// TwinCAT 3 PLC project txi_hxr_motion
// Title: txi-hxr-motion
// Company: SLAC
// ProjectVersion: 2.0.0
// ProgramVersion: 3.1.4024.12
// libraries:
//   LCLS General, * (SLAC)
//   lcls-twincat-motion, * (SLAC)
//   lcls-twincat-physics, * (SLAC)
//   lcls2-cc-lib, * (SLAC)
//   PMPS, * (SLAC - LCLS)
//   Tc2_MC2, * (Beckhoff Automation GmbH)
//   Tc2_Standard, * (Beckhoff Automation GmbH)
//   Tc2_System, * (Beckhoff Automation GmbH)
//   Tc3_Module, * (Beckhoff Automation GmbH)
// project tree:
//   GVLs/ GVL.TcGVL, Main.TcGVL
//   Version/ Global_Version.TcGVL
//   / PlcTask.TcTTO
//   POUs/ PRG_AL1L1_L2SI.TcPOU, PRG_IM2L1_PPM.TcPOU, PRG_01_PLCTASK.TcPOU, PRG_PMPS.TcPOU, PRG_SL3L1_SCATTER.TcPOU, PRG_TXI_PM.TcPOU
//   POUs/temp/ FB_SLITS.TcPOU (not stored), FB_SLITS_POWER.TcPOU (not stored), FB_SLITS_SCATTER.TcPOU (not stored)
// real-time tasks:
//   TASK PlcTask: cycle T#10ms, priority 20, ADS port 350
// motion (NC):
//   TASK NC-Task 1 SAF: cycle T#2ms, priority 4, ADS port 501
//   TASK NC-Task 1 SVB: cycle T#10ms, priority 8, ADS port 511
//   AXIS IM2L1-PPM-MMS (id 2)
//     Dynamic: AccelerationMaximum=200, DecelerationMaximum=200, Acceleration=200, Deceleration=200, Jerk=1000, DelayTime=0.004
//     Velo: Maximum=65
//     MotionControl: Enable=true, Range=0.0005, Time=1
//     TargetPosControl: Range=0.01, Time=1
//     OtherSettings: AllowMotionCmdToSlave=true
//     encoder EncType=29
//       EncPara: ScaleFactorNumerator=5e-05, Offset=-214686.941, MaxCount=#xffffffff, ReferenceSystem=1
//         SoftEndMinControl: Enable=true, Range=-95
//         SoftEndMaxControl: Enable=true, Range=-5
//         Inc: RefSoftSyncMask=#x0000ffff
//     drive DrvType=24
//       Analog: VeloReferenz=100, ScaleFactorActTorque=0.1
//       TimeComp: TaskDelayCycles=1
//     controller CtrType=2
//       CtrPara: PriorControlFactor=1
//         PosDiffControl: Range=10, Time=0.1
//         PID: PosKp=10, PosExtKp=0.01, PosExtVelo=0.0005, DeadBandPosition=0.0001
//         Observer: BandWidth=20
//   AXIS SL3L1-BOTTOM-MMS (id 3)
//   AXIS SL3L1-NORTH-MMS (id 5) // C:\Github\lcls-plc-tmo-motion\plc-tmo-motion\_Config\NC\Axes\SL2K4-NORTH-M25.xti
//     Velo: RefSearch=0.2, RefSync=0.05, Maximum=2.2
//     OtherSettings: AllowMotionCmdToSlave=true
//     encoder EncType=4
//       EncPara: Inverse=true, MaxCount=#x0000ffff
//         SoftEndMinControl: Enable=true, Range=-30.81
//         SoftEndMaxControl: Enable=true
//         Inc: RefSoftSyncMask=#x0000ffff
//     drive DrvType=24
//       Analog: VeloReferenz=2, ScaleFactorActTorque=0.1
//       TimeComp: TaskDelayCycles=1
//     controller CtrType=1
//       CtrPara: PriorControlFactor=1
//         Observer: BandWidth=20
//   AXIS SL3L1-SOUTH-MMS (id 6) // C:\Github\lcls-plc-tmo-motion\plc-tmo-motion\_Config\NC\Axes\SL2K4-SOUTH-M26.xti
//     Velo: RefSearch=0.2, RefSync=0.05, Maximum=2.2
//     OtherSettings: AllowMotionCmdToSlave=true
//     encoder EncType=4
//       EncPara: MaxCount=#x0000ffff
//         SoftEndMinControl: Enable=true, Range=-30.52
//         SoftEndMaxControl: Enable=true
//         Inc: RefSoftSyncMask=#x0000ffff
//     drive DrvType=24
//       Analog: VeloReferenz=2, ScaleFactorActTorque=0.1
//       TimeComp: TaskDelayCycles=1
//     controller CtrType=1
//       CtrPara: PriorControlFactor=1
//         Observer: BandWidth=20
//   AXIS SL3L1-TOP-MMS (id 4) // C:\Github\lcls-plc-tmo-motion\plc-tmo-motion\_Config\NC\Axes\SL2K4-TOP-M24.xti
//     Velo: RefSearch=0.2, RefSync=0.05, Maximum=2.2
//     PositionAreaControl: Range=0.5
//     TargetPosControl: Range=0.1
//     OtherSettings: AllowMotionCmdToSlave=true
//     encoder EncType=4
//       EncPara: Inverse=true, MaxCount=#x0000ffff
//         SoftEndMinControl: Enable=true, Range=-30.91
//         SoftEndMaxControl: Enable=true
//         Inc: RefSoftSyncMask=#x0000ffff
//     drive DrvType=24
//       Analog: VeloReferenz=2, ScaleFactorActTorque=0.1
//       TimeComp: TaskDelayCycles=1
//     controller CtrType=1
//       CtrPara: PriorControlFactor=1
//         PosDiffControl: Range=0.5
//         Observer: BandWidth=20
//   AXIS AL1L1-L2SI-MMS (id 1)
//     Dynamic: AccelerationMaximum=200, DecelerationMaximum=200, Acceleration=200, Deceleration=200, Jerk=500, DelayTime=0.004
//     Velo: Maximum=10
//     TargetPosControl: Range=0.002, Time=2
//     OtherSettings: AllowMotionCmdToSlave=true
//     encoder EncType=29
//       EncPara: ScaleFactorNumerator=5e-05, Offset=-214686.941, MaxCount=#xffffffff, ReferenceSystem=1
//         SoftEndMinControl: Enable=true, Range=-94
//         SoftEndMaxControl: Enable=true, Range=-37
//         Inc: RefSoftSyncMask=#x0000ffff
//     drive DrvType=24
//       Analog: VeloReferenz=100, ScaleFactorActTorque=0.1
//       TimeComp: TaskDelayCycles=1
//     controller CtrType=2
//       CtrPara: PriorControlFactor=1
//         PosDiffControl: Range=1
//         PID: PosKp=20, PosExtKp=1, PosExtVelo=0.1, DeadBandPosition=0.002
//         Observer: BandWidth=20
// I/O:
//   DEVICE Device 1 (EtherCAT), AmsNetId 172.21.136.31.2.1
//     R17-DRL-03 (EK1200) [EK1200-5000 EtherCAT Power supply (2A E-Bus)]
//       Term 8 (EL6070) [EL6070 1Ch. Licensing-Terminal]
//       Term 9 (EL2202) [EL2202 2Ch. Dig. Output 24V, 0.5A]
//       Term 10 (EL6695) [EL6695 EtherCAT Bridge terminal (Primary)]
//       Term 11 (EK1122) [EK1122 2 port EtherCAT junction]
//       Term 12 (EK1110)
//     100H1-L1S01-DRL-02 (EK1100) [EK1100 EtherCAT Coupler (2A E-Bus)]
//       E1 (EK1122) [EK1122 2 port EtherCAT junction]
//         AL1L1-L2SI (EK1100) [EK1100 EtherCAT Coupler (2A E-Bus)]
//           AL1L1-EL7041 [EL7041 1Ch. Stepper motor output stage (50V, 5A)]
//           AL1L1-EL5042 [EL5042 2Ch. BiSS-C Encoder]
//           AL1L1-EL2004 [EL2004 4Ch. Dig. Output 24V, 0.5A]
//           AL1L1-EL4004 [EL4004 4Ch. Ana. Output 0-10V, 12bit]
//           AL1L1-EL9011
//         IM2L1-PPM (EK1100) [EK1100 EtherCAT Coupler (2A E-Bus)]
//           IM2L1-EL7041 [EL7041 1Ch. Stepper motor output stage (50V, 5A)]
//           IM2L1-EL5042 [EL5042 2Ch. BiSS-C Encoder]
//           IM2L1-EL2004
//           IM2L1-EL3314 [EL3314 4Ch. Ana. Input Thermocouple (TC)]
//           IM2L1-EL3052 [EL3052 2Ch. Ana. Input 4-20mA]
//           IM2L1-EL3062 [EL3062 2Ch. Ana. Input 0-10V]
//           IM2L1-EL4004
//           IM2L1-EL9011
//       E2 (EK1122) [EK1122 2 port EtherCAT junction]
//         SL3L1-SCATTER (EK1100) [EK1100 EtherCAT Coupler (2A E-Bus)]
//           SL3L1-EL7031-E1 [EL7031 1Ch. Stepper motor output stage (24V, 1.5A)]
//           SL3L1-EL5101-E2 [EL5101 1Ch. Inc. Encoder 5V]
//           SL3L1-EL7031-E3 [EL7031 1Ch. Stepper motor output stage (24V, 1.5A)]
//           SL3L1-EL5101-E4 [EL5101 1Ch. Inc. Encoder 5V]
//           SL3L1-EL7031-E5 [EL7031 1Ch. Stepper motor output stage (24V, 1.5A)]
//           SL3L1-EL5101-E6
//           SL3L1-EL7031-E7 [EL7031 1Ch. Stepper motor output stage (24V, 1.5A)]
//           SL3L1-EL5101-E8
//           SL3L1-EL9011-E9
//       Term 33 (EK1110) [EK1110 EtherCAT extension]
//     TXI Power Meter (EK1100) [EK1100 EtherCAT Coupler (2A E-Bus)]
//       PM-EL3064
//       Term 70 (EK1122) [EK1122 2 port EtherCAT junction]
//       Term 74 (EL9011) [EL9011 End Terminal]
// variable links:
//   (this object) <-> Device 1 (EtherCAT)/100H1-L1S01-DRL-02 (EK1100)/E1 (EK1122)/IM2L1-PPM (EK1100)/IM2L1-EL5042
//     Enc/Inputs/In/nComState @bit 1 <-> WcState/InputToggle
//     Enc/Inputs/In/nComState <-> WcState/WcState
//     Enc/Inputs/In/nDataIn1 <-> FB Inputs Channel 1/Position
//     Enc/Inputs/In/nState1 @bit 12 <-> FB Inputs Channel 1/Status/Diag
//     Enc/Inputs/In/nState1 @bit 1 <-> FB Inputs Channel 1/Status/Error
//     Enc/Inputs/In/nState1 @bit 14 <-> FB Inputs Channel 1/Status/Input cycle counter
//     Enc/Inputs/In/nState1 @bit 2 <-> FB Inputs Channel 1/Status/Ready
//     Enc/Inputs/In/nState1 @bit 13 <-> FB Inputs Channel 1/Status/TxPDO State
//     Enc/Inputs/In/nState1 <-> FB Inputs Channel 1/Status/Warning
//   (this object) <-> Device 1 (EtherCAT)/100H1-L1S01-DRL-02 (EK1100)/E1 (EK1122)/IM2L1-PPM (EK1100)/IM2L1-EL7041
//     Drive/Inputs/In/nState1 @bit 3 <-> STM Status/Status/Error
//     Drive/Inputs/In/nState1 @bit 5 <-> STM Status/Status/Moving negative
//     Drive/Inputs/In/nState1 @bit 4 <-> STM Status/Status/Moving positive
//     Drive/Inputs/In/nState1 @bit 1 <-> STM Status/Status/Ready
//     Drive/Inputs/In/nState1 <-> STM Status/Status/Ready to enable
//     Drive/Inputs/In/nState1 @bit 6 <-> STM Status/Status/Torque reduced
//     Drive/Inputs/In/nState1 @bit 2 <-> STM Status/Status/Warning
//     Drive/Inputs/In/nState2 @bit 3 <-> STM Status/Status/Digital input 1
//     Drive/Inputs/In/nState2 @bit 4 <-> STM Status/Status/Digital input 2
//     Drive/Inputs/In/nState2 @bit 5 <-> STM Status/Status/Sync error
//     Drive/Inputs/In/nState2 @bit 7 <-> STM Status/Status/TxPDO Toggle
//     Drive/Inputs/In/nState4 @bit 1 <-> WcState/InputToggle
//     Drive/Inputs/In/nState4 <-> WcState/WcState
//     Drive/Outputs/Out/nCtrl1 <-> STM Control/Control/Enable
//     Drive/Outputs/Out/nCtrl1 @bit 2 <-> STM Control/Control/Reduce torque
//     Drive/Outputs/Out/nCtrl1 @bit 1 <-> STM Control/Control/Reset
//     Drive/Outputs/Out/nDataOut2[0] <-> STM Velocity/Velocity
//   (this object) <-> Device 1 (EtherCAT)/100H1-L1S01-DRL-02 (EK1100)/E2 (EK1122)/SL3L1-SCATTER (EK1100)/SL3L1-EL5101-E6
//     Enc/Inputs/In/nDataIn1[0] <-> ENC Status compact/Counter value
//     Enc/Inputs/In/nDataIn2[0] <-> ENC Status compact/Latch value
//     Enc/Inputs/In/nState1 @bit 4 <-> ENC Status compact/Status/Counter overflow
//     Enc/Inputs/In/nState1 @bit 3 <-> ENC Status compact/Status/Counter underflow
//     Enc/Inputs/In/nState1 @bit 7 <-> ENC Status compact/Status/Extrapolation stall
//     Enc/Inputs/In/nState1 <-> ENC Status compact/Status/Latch C valid
//     Enc/Inputs/In/nState1 @bit 1 <-> ENC Status compact/Status/Latch extern valid
//     Enc/Inputs/In/nState1 @bit 6 <-> ENC Status compact/Status/Open circuit
//     Enc/Inputs/In/nState1 @bit 2 <-> ENC Status compact/Status/Set counter done
//     Enc/Inputs/In/nState1 @bit 5 <-> ENC Status compact/Status/Status of input status
//     Enc/Inputs/In/nState2 @bit 4 <-> ENC Status compact/Status/Status of extern latch
//     Enc/Inputs/In/nState2 <-> ENC Status compact/Status/Status of input A
//     Enc/Inputs/In/nState2 @bit 1 <-> ENC Status compact/Status/Status of input B
//     Enc/Inputs/In/nState2 @bit 2 <-> ENC Status compact/Status/Status of input C
//     Enc/Inputs/In/nState2 @bit 3 <-> ENC Status compact/Status/Status of input gate
//     Enc/Inputs/In/nState2 @bit 5 <-> ENC Status compact/Status/Sync error
//     Enc/Inputs/In/nState2 @bit 6 <-> ENC Status compact/Status/TxPDO State
//     Enc/Inputs/In/nState2 @bit 7 <-> ENC Status compact/Status/TxPDO Toggle
//     Enc/Inputs/In/nState4 @bit 1 <-> WcState/InputToggle
//     Enc/Inputs/In/nState4 <-> WcState/WcState
//     Enc/Outputs/Out/nCtrl1 <-> ENC Control compact/Control/Enable latch C
//     Enc/Outputs/Out/nCtrl1 @bit 3 <-> ENC Control compact/Control/Enable latch extern on negative edge
//     Enc/Outputs/Out/nCtrl1 @bit 1 <-> ENC Control compact/Control/Enable latch extern on positive edge
//     Enc/Outputs/Out/nCtrl1 @bit 2 <-> ENC Control compact/Control/Set counter
//     Enc/Outputs/Out/nDataOut1[0] <-> ENC Control compact/Set counter value
//   (this object) <-> Device 1 (EtherCAT)/100H1-L1S01-DRL-02 (EK1100)/E2 (EK1122)/SL3L1-SCATTER (EK1100)/SL3L1-EL7031-E5
//     Drive/Inputs/In/nState1 @bit 3 <-> STM Status/Status/Error
//     Drive/Inputs/In/nState1 @bit 5 <-> STM Status/Status/Moving negative
//     Drive/Inputs/In/nState1 @bit 4 <-> STM Status/Status/Moving positive
//     Drive/Inputs/In/nState1 @bit 1 <-> STM Status/Status/Ready
//     Drive/Inputs/In/nState1 <-> STM Status/Status/Ready to enable
//     Drive/Inputs/In/nState1 @bit 6 <-> STM Status/Status/Torque reduced
//     Drive/Inputs/In/nState1 @bit 2 <-> STM Status/Status/Warning
//     Drive/Inputs/In/nState2 @bit 3 <-> STM Status/Status/Digital input 1
//     Drive/Inputs/In/nState2 @bit 4 <-> STM Status/Status/Digital input 2
//     Drive/Inputs/In/nState2 @bit 5 <-> STM Status/Status/Sync error
//     Drive/Inputs/In/nState2 @bit 7 <-> STM Status/Status/TxPDO Toggle
//     Drive/Inputs/In/nState4 @bit 1 <-> WcState/InputToggle
//     Drive/Inputs/In/nState4 <-> WcState/WcState
//     Drive/Outputs/Out/nCtrl1 <-> STM Control/Control/Enable
//     Drive/Outputs/Out/nCtrl1 @bit 2 <-> STM Control/Control/Reduce torque
//     Drive/Outputs/Out/nCtrl1 @bit 1 <-> STM Control/Control/Reset
//     Drive/Outputs/Out/nDataOut2[0] <-> STM Velocity/Velocity
//   (this object) <-> Device 1 (EtherCAT)/100H1-L1S01-DRL-02 (EK1100)/E2 (EK1122)/SL3L1-SCATTER (EK1100)/SL3L1-EL5101-E8
//     Enc/Inputs/In/nDataIn1[0] <-> ENC Status compact/Counter value
//     Enc/Inputs/In/nDataIn2[0] <-> ENC Status compact/Latch value
//     Enc/Inputs/In/nState1 @bit 4 <-> ENC Status compact/Status/Counter overflow
//     Enc/Inputs/In/nState1 @bit 3 <-> ENC Status compact/Status/Counter underflow
//     Enc/Inputs/In/nState1 @bit 7 <-> ENC Status compact/Status/Extrapolation stall
//     Enc/Inputs/In/nState1 <-> ENC Status compact/Status/Latch C valid
//     Enc/Inputs/In/nState1 @bit 1 <-> ENC Status compact/Status/Latch extern valid
//     Enc/Inputs/In/nState1 @bit 6 <-> ENC Status compact/Status/Open circuit
//     Enc/Inputs/In/nState1 @bit 2 <-> ENC Status compact/Status/Set counter done
//     Enc/Inputs/In/nState1 @bit 5 <-> ENC Status compact/Status/Status of input status
//     Enc/Inputs/In/nState2 @bit 4 <-> ENC Status compact/Status/Status of extern latch
//     Enc/Inputs/In/nState2 <-> ENC Status compact/Status/Status of input A
//     Enc/Inputs/In/nState2 @bit 1 <-> ENC Status compact/Status/Status of input B
//     Enc/Inputs/In/nState2 @bit 2 <-> ENC Status compact/Status/Status of input C
//     Enc/Inputs/In/nState2 @bit 3 <-> ENC Status compact/Status/Status of input gate
//     Enc/Inputs/In/nState2 @bit 5 <-> ENC Status compact/Status/Sync error
//     Enc/Inputs/In/nState2 @bit 6 <-> ENC Status compact/Status/TxPDO State
//     Enc/Inputs/In/nState2 @bit 7 <-> ENC Status compact/Status/TxPDO Toggle
//     Enc/Inputs/In/nState4 @bit 1 <-> WcState/InputToggle
//     Enc/Inputs/In/nState4 <-> WcState/WcState
//     Enc/Outputs/Out/nCtrl1 <-> ENC Control compact/Control/Enable latch C
//     Enc/Outputs/Out/nCtrl1 @bit 3 <-> ENC Control compact/Control/Enable latch extern on negative edge
//     Enc/Outputs/Out/nCtrl1 @bit 1 <-> ENC Control compact/Control/Enable latch extern on positive edge
//     Enc/Outputs/Out/nCtrl1 @bit 2 <-> ENC Control compact/Control/Set counter
//     Enc/Outputs/Out/nDataOut1[0] <-> ENC Control compact/Set counter value
//   (this object) <-> Device 1 (EtherCAT)/100H1-L1S01-DRL-02 (EK1100)/E2 (EK1122)/SL3L1-SCATTER (EK1100)/SL3L1-EL7031-E7
//     Drive/Inputs/In/nState1 @bit 3 <-> STM Status/Status/Error
//     Drive/Inputs/In/nState1 @bit 5 <-> STM Status/Status/Moving negative
//     Drive/Inputs/In/nState1 @bit 4 <-> STM Status/Status/Moving positive
//     Drive/Inputs/In/nState1 @bit 1 <-> STM Status/Status/Ready
//     Drive/Inputs/In/nState1 <-> STM Status/Status/Ready to enable
//     Drive/Inputs/In/nState1 @bit 6 <-> STM Status/Status/Torque reduced
//     Drive/Inputs/In/nState1 @bit 2 <-> STM Status/Status/Warning
//     Drive/Inputs/In/nState2 @bit 3 <-> STM Status/Status/Digital input 1
//     Drive/Inputs/In/nState2 @bit 4 <-> STM Status/Status/Digital input 2
//     Drive/Inputs/In/nState2 @bit 5 <-> STM Status/Status/Sync error
//     Drive/Inputs/In/nState2 @bit 7 <-> STM Status/Status/TxPDO Toggle
//     Drive/Inputs/In/nState4 @bit 1 <-> WcState/InputToggle
//     Drive/Inputs/In/nState4 <-> WcState/WcState
//     Drive/Outputs/Out/nCtrl1 <-> STM Control/Control/Enable
//     Drive/Outputs/Out/nCtrl1 @bit 2 <-> STM Control/Control/Reduce torque
//     Drive/Outputs/Out/nCtrl1 @bit 1 <-> STM Control/Control/Reset
//     Drive/Outputs/Out/nDataOut2[0] <-> STM Velocity/Velocity
//   (this object) <-> Device 1 (EtherCAT)/100H1-L1S01-DRL-02 (EK1100)/E2 (EK1122)/SL3L1-SCATTER (EK1100)/SL3L1-EL5101-E4
//     Enc/Inputs/In/nDataIn1[0] <-> ENC Status compact/Counter value
//     Enc/Inputs/In/nDataIn2[0] <-> ENC Status compact/Latch value
//     Enc/Inputs/In/nState1 @bit 4 <-> ENC Status compact/Status/Counter overflow
//     Enc/Inputs/In/nState1 @bit 3 <-> ENC Status compact/Status/Counter underflow
//     Enc/Inputs/In/nState1 @bit 7 <-> ENC Status compact/Status/Extrapolation stall
//     Enc/Inputs/In/nState1 <-> ENC Status compact/Status/Latch C valid
//     Enc/Inputs/In/nState1 @bit 1 <-> ENC Status compact/Status/Latch extern valid
//     Enc/Inputs/In/nState1 @bit 6 <-> ENC Status compact/Status/Open circuit
//     Enc/Inputs/In/nState1 @bit 2 <-> ENC Status compact/Status/Set counter done
//     Enc/Inputs/In/nState1 @bit 5 <-> ENC Status compact/Status/Status of input status
//     Enc/Inputs/In/nState2 @bit 4 <-> ENC Status compact/Status/Status of extern latch
//     Enc/Inputs/In/nState2 <-> ENC Status compact/Status/Status of input A
//     Enc/Inputs/In/nState2 @bit 1 <-> ENC Status compact/Status/Status of input B
//     Enc/Inputs/In/nState2 @bit 2 <-> ENC Status compact/Status/Status of input C
//     Enc/Inputs/In/nState2 @bit 3 <-> ENC Status compact/Status/Status of input gate
//     Enc/Inputs/In/nState2 @bit 5 <-> ENC Status compact/Status/Sync error
//     Enc/Inputs/In/nState2 @bit 6 <-> ENC Status compact/Status/TxPDO State
//     Enc/Inputs/In/nState2 @bit 7 <-> ENC Status compact/Status/TxPDO Toggle
//     Enc/Inputs/In/nState4 @bit 1 <-> WcState/InputToggle
//     Enc/Inputs/In/nState4 <-> WcState/WcState
//     Enc/Outputs/Out/nCtrl1 <-> ENC Control compact/Control/Enable latch C
//     Enc/Outputs/Out/nCtrl1 @bit 3 <-> ENC Control compact/Control/Enable latch extern on negative edge
//     Enc/Outputs/Out/nCtrl1 @bit 1 <-> ENC Control compact/Control/Enable latch extern on positive edge
//     Enc/Outputs/Out/nCtrl1 @bit 2 <-> ENC Control compact/Control/Set counter
//     Enc/Outputs/Out/nDataOut1[0] <-> ENC Control compact/Set counter value
//   (this object) <-> Device 1 (EtherCAT)/100H1-L1S01-DRL-02 (EK1100)/E2 (EK1122)/SL3L1-SCATTER (EK1100)/SL3L1-EL7031-E3
//     Drive/Inputs/In/nState1 @bit 3 <-> STM Status/Status/Error
//     Drive/Inputs/In/nState1 @bit 5 <-> STM Status/Status/Moving negative
//     Drive/Inputs/In/nState1 @bit 4 <-> STM Status/Status/Moving positive
//     Drive/Inputs/In/nState1 @bit 1 <-> STM Status/Status/Ready
//     Drive/Inputs/In/nState1 <-> STM Status/Status/Ready to enable
//     Drive/Inputs/In/nState1 @bit 6 <-> STM Status/Status/Torque reduced
//     Drive/Inputs/In/nState1 @bit 2 <-> STM Status/Status/Warning
//     Drive/Inputs/In/nState2 @bit 3 <-> STM Status/Status/Digital input 1
//     Drive/Inputs/In/nState2 @bit 4 <-> STM Status/Status/Digital input 2
//     Drive/Inputs/In/nState2 @bit 5 <-> STM Status/Status/Sync error
//     Drive/Inputs/In/nState2 @bit 7 <-> STM Status/Status/TxPDO Toggle
//     Drive/Inputs/In/nState4 @bit 1 <-> WcState/InputToggle
//     Drive/Inputs/In/nState4 <-> WcState/WcState
//     Drive/Outputs/Out/nCtrl1 <-> STM Control/Control/Enable
//     Drive/Outputs/Out/nCtrl1 @bit 2 <-> STM Control/Control/Reduce torque
//     Drive/Outputs/Out/nCtrl1 @bit 1 <-> STM Control/Control/Reset
//     Drive/Outputs/Out/nDataOut2[0] <-> STM Velocity/Velocity
//   (this object) <-> Device 1 (EtherCAT)/100H1-L1S01-DRL-02 (EK1100)/E1 (EK1122)/AL1L1-L2SI (EK1100)/AL1L1-EL5042
//     Enc/Inputs/In/nComState @bit 1 <-> WcState/InputToggle
//     Enc/Inputs/In/nComState <-> WcState/WcState
//     Enc/Inputs/In/nDataIn1 <-> FB Inputs Channel 1/Position
//     Enc/Inputs/In/nState1 @bit 12 <-> FB Inputs Channel 1/Status/Diag
//     Enc/Inputs/In/nState1 @bit 1 <-> FB Inputs Channel 1/Status/Error
//     Enc/Inputs/In/nState1 @bit 14 <-> FB Inputs Channel 1/Status/Input cycle counter
//     Enc/Inputs/In/nState1 @bit 2 <-> FB Inputs Channel 1/Status/Ready
//     Enc/Inputs/In/nState1 @bit 13 <-> FB Inputs Channel 1/Status/TxPDO State
//     Enc/Inputs/In/nState1 <-> FB Inputs Channel 1/Status/Warning
//   (this object) <-> Device 1 (EtherCAT)/100H1-L1S01-DRL-02 (EK1100)/E1 (EK1122)/AL1L1-L2SI (EK1100)/AL1L1-EL7041
//     Drive/Inputs/In/nState1 @bit 3 <-> STM Status/Status/Error
//     Drive/Inputs/In/nState1 @bit 5 <-> STM Status/Status/Moving negative
//     Drive/Inputs/In/nState1 @bit 4 <-> STM Status/Status/Moving positive
//     Drive/Inputs/In/nState1 @bit 1 <-> STM Status/Status/Ready
//     Drive/Inputs/In/nState1 <-> STM Status/Status/Ready to enable
//     Drive/Inputs/In/nState1 @bit 6 <-> STM Status/Status/Torque reduced
//     Drive/Inputs/In/nState1 @bit 2 <-> STM Status/Status/Warning
//     Drive/Inputs/In/nState2 @bit 3 <-> STM Status/Status/Digital input 1
//     Drive/Inputs/In/nState2 @bit 4 <-> STM Status/Status/Digital input 2
//     Drive/Inputs/In/nState2 @bit 5 <-> STM Status/Status/Sync error
//     Drive/Inputs/In/nState2 @bit 7 <-> STM Status/Status/TxPDO Toggle
//     Drive/Inputs/In/nState4 @bit 1 <-> WcState/InputToggle
//     Drive/Inputs/In/nState4 <-> WcState/WcState
//     Drive/Outputs/Out/nCtrl1 <-> STM Control/Control/Enable
//     Drive/Outputs/Out/nCtrl1 @bit 2 <-> STM Control/Control/Reduce torque
//     Drive/Outputs/Out/nCtrl1 @bit 1 <-> STM Control/Control/Reset
//     Drive/Outputs/Out/nDataOut2[0] <-> STM Velocity/Velocity
//   txi_hxr_motion Instance <-> Device 1 (EtherCAT)/100H1-L1S01-DRL-02 (EK1100)/E1 (EK1122)/AL1L1-L2SI (EK1100)/AL1L1-EL2004
//     PlcTask Outputs/Main.M1.bBrakeRelease <-> Channel 1/Output
//   txi_hxr_motion Instance <-> Device 1 (EtherCAT)/100H1-L1S01-DRL-02 (EK1100)/E1 (EK1122)/AL1L1-L2SI (EK1100)/AL1L1-EL4004
//     PlcTask Outputs/PRG_AL1L1_L2SI.fbAL1L1.fbLaser.iLaserINT <-> AO Outputs Channel 1/Analog output
//     PlcTask Outputs/PRG_AL1L1_L2SI.fbAL1L1.fbLaser.iShutdownINT <-> AO Outputs Channel 2/Analog output
//   txi_hxr_motion Instance <-> Device 1 (EtherCAT)/100H1-L1S01-DRL-02 (EK1100)/E1 (EK1122)/AL1L1-L2SI (EK1100)/AL1L1-EL5042
//     PlcTask Inputs/Main.M1.nRawEncoderULINT <-> FB Inputs Channel 1/Position
//   txi_hxr_motion Instance <-> Device 1 (EtherCAT)/100H1-L1S01-DRL-02 (EK1100)/E1 (EK1122)/AL1L1-L2SI (EK1100)/AL1L1-EL7041
//     PlcTask Inputs/Main.M1.bLimitBackwardEnable <-> STM Status/Status/Digital input 2
//     PlcTask Inputs/Main.M1.bLimitForwardEnable <-> STM Status/Status/Digital input 1
//   txi_hxr_motion Instance <-> Device 1 (EtherCAT)/100H1-L1S01-DRL-02 (EK1100)/E1 (EK1122)/IM2L1-PPM (EK1100)/IM2L1-EL2004
//     PlcTask Outputs/Main.M2.bBrakeRelease <-> Channel 1/Output
//     PlcTask Outputs/PRG_IM2L1_PPM.fbIM2L1.fbGige.bGigePower <-> Channel 3/Output
//   txi_hxr_motion Instance <-> Device 1 (EtherCAT)/100H1-L1S01-DRL-02 (EK1100)/E1 (EK1122)/IM2L1-PPM (EK1100)/IM2L1-EL3062
//     PlcTask Inputs/PRG_IM2L1_PPM.fbIM2L1.fbPowerMeter.iVoltageINT <-> AI Standard Channel 1/Value
//   txi_hxr_motion Instance <-> Device 1 (EtherCAT)/100H1-L1S01-DRL-02 (EK1100)/E1 (EK1122)/IM2L1-PPM (EK1100)/IM2L1-EL3314
//     PlcTask Inputs/PRG_IM2L1_PPM.fbIM2L1.fbPowerMeter.fbThermoCouple.bError <-> TC Inputs Channel 1/Status/Error
//     PlcTask Inputs/PRG_IM2L1_PPM.fbIM2L1.fbPowerMeter.fbThermoCouple.bOverrange <-> TC Inputs Channel 1/Status/Overrange
//     PlcTask Inputs/PRG_IM2L1_PPM.fbIM2L1.fbPowerMeter.fbThermoCouple.bUnderrange <-> TC Inputs Channel 1/Status/Underrange
//     PlcTask Inputs/PRG_IM2L1_PPM.fbIM2L1.fbPowerMeter.fbThermoCouple.iRaw <-> TC Inputs Channel 1/Value
//     PlcTask Inputs/PRG_IM2L1_PPM.fbIM2L1.fbYagThermoCouple.bError <-> TC Inputs Channel 2/Status/Error
//     PlcTask Inputs/PRG_IM2L1_PPM.fbIM2L1.fbYagThermoCouple.bOverrange <-> TC Inputs Channel 2/Status/Overrange
//     PlcTask Inputs/PRG_IM2L1_PPM.fbIM2L1.fbYagThermoCouple.bUnderrange <-> TC Inputs Channel 2/Status/Underrange
//     PlcTask Inputs/PRG_IM2L1_PPM.fbIM2L1.fbYagThermoCouple.iRaw <-> TC Inputs Channel 2/Value
//   txi_hxr_motion Instance <-> Device 1 (EtherCAT)/100H1-L1S01-DRL-02 (EK1100)/E1 (EK1122)/IM2L1-PPM (EK1100)/IM2L1-EL4004
//     PlcTask Outputs/PRG_IM2L1_PPM.fbIM2L1.fbGige.iIlluminatorINT <-> AO Outputs Channel 1/Analog output
//   txi_hxr_motion Instance <-> Device 1 (EtherCAT)/100H1-L1S01-DRL-02 (EK1100)/E1 (EK1122)/IM2L1-PPM (EK1100)/IM2L1-EL7041
//     PlcTask Inputs/Main.M2.bLimitBackwardEnable <-> STM Status/Status/Digital input 2
//     PlcTask Inputs/Main.M2.bLimitForwardEnable <-> STM Status/Status/Digital input 1
//   txi_hxr_motion Instance <-> Device 1 (EtherCAT)/100H1-L1S01-DRL-02 (EK1100)/E2 (EK1122)/SL3L1-SCATTER (EK1100)/SL3L1-EL5101-E2
//     PlcTask Inputs/Main.M3.nRawEncoderUINT <-> ENC Status compact/Counter value
//   txi_hxr_motion Instance <-> Device 1 (EtherCAT)/100H1-L1S01-DRL-02 (EK1100)/E2 (EK1122)/SL3L1-SCATTER (EK1100)/SL3L1-EL5101-E4
//     PlcTask Inputs/Main.M4.nRawEncoderUINT <-> ENC Status compact/Counter value
//   txi_hxr_motion Instance <-> Device 1 (EtherCAT)/100H1-L1S01-DRL-02 (EK1100)/E2 (EK1122)/SL3L1-SCATTER (EK1100)/SL3L1-EL5101-E6
//     PlcTask Inputs/Main.M5.nRawEncoderUINT <-> ENC Status compact/Counter value
//   txi_hxr_motion Instance <-> Device 1 (EtherCAT)/100H1-L1S01-DRL-02 (EK1100)/E2 (EK1122)/SL3L1-SCATTER (EK1100)/SL3L1-EL5101-E8
//     PlcTask Inputs/Main.M6.nRawEncoderUINT <-> ENC Status compact/Counter value
//   txi_hxr_motion Instance <-> Device 1 (EtherCAT)/100H1-L1S01-DRL-02 (EK1100)/E2 (EK1122)/SL3L1-SCATTER (EK1100)/SL3L1-EL7031-E1
//     PlcTask Inputs/Main.M3.bLimitBackwardEnable <-> STM Status/Status/Digital input 1
//     PlcTask Inputs/Main.M3.bLimitForwardEnable <-> STM Status/Status/Digital input 2
//   txi_hxr_motion Instance <-> Device 1 (EtherCAT)/100H1-L1S01-DRL-02 (EK1100)/E2 (EK1122)/SL3L1-SCATTER (EK1100)/SL3L1-EL7031-E3
//     PlcTask Inputs/Main.M4.bLimitBackwardEnable <-> STM Status/Status/Digital input 1
//     PlcTask Inputs/Main.M4.bLimitForwardEnable <-> STM Status/Status/Digital input 2
//   txi_hxr_motion Instance <-> Device 1 (EtherCAT)/100H1-L1S01-DRL-02 (EK1100)/E2 (EK1122)/SL3L1-SCATTER (EK1100)/SL3L1-EL7031-E5
//     PlcTask Inputs/Main.M5.bLimitBackwardEnable <-> STM Status/Status/Digital input 2
//     PlcTask Inputs/Main.M5.bLimitForwardEnable <-> STM Status/Status/Digital input 1
//   txi_hxr_motion Instance <-> Device 1 (EtherCAT)/100H1-L1S01-DRL-02 (EK1100)/E2 (EK1122)/SL3L1-SCATTER (EK1100)/SL3L1-EL7031-E7
//     PlcTask Inputs/Main.M6.bLimitBackwardEnable <-> STM Status/Status/Digital input 2
//     PlcTask Inputs/Main.M6.bLimitForwardEnable <-> STM Status/Status/Digital input 1
//   txi_hxr_motion Instance <-> Device 1 (EtherCAT)/R17-DRL-03 (EK1200)/PMPS_FFO
//     PlcTask Outputs/GVL.fbFastFaultOutput1.q_xFastFaultOut <-> Channel 1/Output
//   txi_hxr_motion Instance <-> Device 1 (EtherCAT)/R17-DRL-03 (EK1200)/PMPS_PRE
//     PlcTask Inputs/PRG_PMPS.fbArbiterIO.i_stCurrentBP <-> IO Inputs/CurrentBP
//     PlcTask Inputs/PRG_PMPS.fbArbiterIO.xTxPDO_state <-> SYNC Inputs/TxPDO state
//     PlcTask Inputs/PRG_PMPS.fbArbiterIO.xTxPDO_toggle <-> SYNC Inputs/TxPDO toggle
//     PlcTask Outputs/PRG_PMPS.fbArbiterIO.q_stRequestedBP <-> IO Outputs/RequestedBP
//   txi_hxr_motion Instance <-> Device 1 (EtherCAT)/TXI Power Meter (EK1100)/PM-EL3064
//     PlcTask Inputs/PRG_TXI_PM.fbTXIPM.fbPowerMeter.iVoltageINT <-> AI Standard Channel 1/Value
//   txi_hxr_motion Instance <-> NC-Task 1 SAF/Axes/AL1L1-L2SI-MMS
//     PlcTask Inputs/Main.M1.Axis.NcToPlc <-> Outputs/ToPlc
//     PlcTask Outputs/Main.M1.Axis.PlcToNc <-> Inputs/FromPlc
//   txi_hxr_motion Instance <-> NC-Task 1 SAF/Axes/IM2L1-PPM-MMS
//     PlcTask Inputs/Main.M2.Axis.NcToPlc <-> Outputs/ToPlc
//     PlcTask Outputs/Main.M2.Axis.PlcToNc <-> Inputs/FromPlc
//   txi_hxr_motion Instance <-> NC-Task 1 SAF/Axes/SL3L1-BOTTOM-MMS
//     PlcTask Inputs/Main.M3.Axis.NcToPlc <-> Outputs/ToPlc
//     PlcTask Outputs/Main.M3.Axis.PlcToNc <-> Inputs/FromPlc
//   txi_hxr_motion Instance <-> NC-Task 1 SAF/Axes/SL3L1-NORTH-MMS
//     PlcTask Inputs/Main.M5.Axis.NcToPlc <-> Outputs/ToPlc
//     PlcTask Outputs/Main.M5.Axis.PlcToNc <-> Inputs/FromPlc
//   txi_hxr_motion Instance <-> NC-Task 1 SAF/Axes/SL3L1-SOUTH-MMS
//     PlcTask Inputs/Main.M6.Axis.NcToPlc <-> Outputs/ToPlc
//     PlcTask Outputs/Main.M6.Axis.PlcToNc <-> Inputs/FromPlc
//   txi_hxr_motion Instance <-> NC-Task 1 SAF/Axes/SL3L1-TOP-MMS
//     PlcTask Inputs/Main.M4.Axis.NcToPlc <-> Outputs/ToPlc
//     PlcTask Outputs/Main.M4.Axis.PlcToNc <-> Inputs/FromPlc

CONFIGURATION txi_hxr_motion
    RESOURCE PLC ON TwinCAT3
        TASK PlcTask(INTERVAL := T#10ms, PRIORITY := 20);
        PROGRAM PRG_01_PLCTASK WITH PlcTask : PRG_01_PLCTASK;
    END_RESOURCE
END_CONFIGURATION

// ---- GVLs/GVL.TcGVL
{attribute 'qualified_only'}
VAR_GLOBAL
    {attribute 'pytmc' := 'pv: PLC:TXI:MOTION:ARB:01'}
    fbArbiter1: FB_Arbiter(1);

    // For all devices after Stopper
    {attribute 'pytmc' := 'pv: PLC:TXI:MOTION:FFO:01'}
    {attribute 'TcLinkTo' := '.q_xFastFaultOut:=TIIB[PMPS_FFO]^Channel 1^Output'}
    fbFastFaultOutput1: FB_HardwareFFOutput := (bAutoReset := TRUE, i_sNetID:='');

END_VAR

// ---- Version/Global_Version.TcGVL
{attribute 'TcGenerated'}
{attribute 'no-analysis'}
{attribute 'linkalways'}
// This function has been automatically generated from the project information.
VAR_GLOBAL CONSTANT
    {attribute 'const_non_replaced'}
    stLibVersion_txi_hxr_motion : ST_LibVersion := (iMajor := 2, iMinor := 0, iBuild := 0, iRevision := 0, nFlags := 1, sVersion := '2.0.0');
END_VAR

// ---- GVLs/Main.TcGVL
{attribute 'qualified_only'}
VAR_GLOBAL
     // AL1L1-L2SI
    {attribute 'pytmc' := 'pv: AL1L1:L2SI:MMS'}
    {attribute 'TcLinkTo' := '.bLimitForwardEnable  := TIIB[AL1L1-EL7041]^STM Status^Status^Digital input 1;
                              .bLimitBackwardEnable := TIIB[AL1L1-EL7041]^STM Status^Status^Digital input 2;
                              .bBrakeRelease        := TIIB[AL1L1-EL2004]^Channel 1^Output;
                              .nRawEncoderULINT     := TIIB[AL1L1-EL5042]^FB Inputs Channel 1^Position'}
    M1: DUT_MotionStage := (sName := 'AL1L1:L2SI:MMS');

    // IM2L1-PPM-MMS
    {attribute 'pytmc' := 'pv: IM2L1:PPM:MMS'}
    {attribute 'TcLinkTo' := '.bLimitForwardEnable  := TIIB[IM2L1-EL7041]^STM Status^Status^Digital input 1;
                              .bLimitBackwardEnable := TIIB[IM2L1-EL7041]^STM Status^Status^Digital input 2;
                              .bBrakeRelease        := TIIB[IM2L1-EL2004]^Channel 1^Output'}
    M2: DUT_MotionStage := (sName := 'IM2L1:PPM:MMS');

    //SL3L1-SCATTER: 4 Axes
    {attribute 'pytmc' := 'pv: SL3L1:SCATTER:MMS:BOTTOM'}
    {attribute 'TcLinkTo' := '.bLimitForwardEnable  := TIIB[SL3L1-EL7031-E1]^STM Status^Status^Digital input 2;
                              .bLimitBackwardEnable := TIIB[SL3L1-EL7031-E1]^STM Status^Status^Digital input 1;
                              .nRawEncoderUINT      := TIIB[SL3L1-EL5101-E2]^ENC Status compact^Counter value'}
    M3: DUT_MotionStage := (sName := 'SL3L1:SCATTER:MMS:BOTTOM');
    {attribute 'pytmc' := 'pv: SL3L1:SCATTER:MMS:TOP'}
    {attribute 'TcLinkTo' := '.bLimitForwardEnable  := TIIB[SL3L1-EL7031-E3]^STM Status^Status^Digital input 2;
                              .bLimitBackwardEnable := TIIB[SL3L1-EL7031-E3]^STM Status^Status^Digital input 1;
                              .nRawEncoderUINT      := TIIB[SL3L1-EL5101-E4]^ENC Status compact^Counter value'}
    M4: DUT_MotionStage := (sName := 'SL3L1:SCATTER:MMS:TOP');
    {attribute 'pytmc' := 'pv: SL3L1:SCATTER:MMS:NORTH'}
    {attribute 'TcLinkTo' := '.bLimitForwardEnable  := TIIB[SL3L1-EL7031-E5]^STM Status^Status^Digital input 1;
                              .bLimitBackwardEnable := TIIB[SL3L1-EL7031-E5]^STM Status^Status^Digital input 2;
                              .nRawEncoderUINT      := TIIB[SL3L1-EL5101-E6]^ENC Status compact^Counter value'}
    M5: DUT_MotionStage := (sName := 'SL3L1:SCATTER:MMS:NORTH');
    {attribute 'pytmc' := 'pv: SL3L1:SCATTER:MMS:SOUTH'}
    {attribute 'TcLinkTo' := '.bLimitForwardEnable  := TIIB[SL3L1-EL7031-E7]^STM Status^Status^Digital input 1;
                              .bLimitBackwardEnable := TIIB[SL3L1-EL7031-E7]^STM Status^Status^Digital input 2;
                              .nRawEncoderUINT      := TIIB[SL3L1-EL5101-E8]^ENC Status compact^Counter value'}
    M6: DUT_MotionStage := (sName := 'SL3L1:SCATTER:MMS:SOUTH');
END_VAR

// ---- POUs/PRG_01_PLCTASK.TcPOU
PROGRAM PRG_01_PLCTASK
VAR
    fbLogHandler: FB_LogHandler;
END_VAR

PRG_AL1L1_L2SI();
PRG_IM2L1_PPM();
PRG_SL3L1_SCATTER();
PRG_TXI_PM();
PRG_PMPS();
fbLogHandler();

END_PROGRAM

// ---- POUs/PRG_AL1L1_L2SI.TcPOU
PROGRAM PRG_AL1L1_L2SI
VAR
    {attribute 'pytmc' := '
        pv: AL1L1:L2SI
        io: io
    '}
    {attribute 'TcLinkTo' := '.fbLaser.iLaserINT := TIIB[AL1L1-EL4004]^AO Outputs Channel 1^Analog output;
                              .fbLaser.iShutdownINT := TIIB[AL1L1-EL4004]^AO Outputs Channel 2^Analog output'}
    fbAL1L1: FB_REF;
END_VAR

//fbAL1L1.nTransitionAssertionID := 16#6120;
//fbAL1L1.nUnknownAssertionID := 16#6129;

fbAL1L1.stOut.fPosition := -38.0; // Upper limit
fbAL1L1.stOut.bUseRawCounts := FALSE;
//fbAL1L1.stOut.nRequestAssertionID := 16#6121;
//fbAL1L1.stOut.stBeamParams := PMPS_GVL.cstFullBeam;
fbAL1L1.stOut.bValid := TRUE;

fbAL1L1.stIn.fPosition := -90.0; // Current position at time of edit
fbAL1L1.stIn.bUseRawCounts := FALSE;
//fbAL1L1.stIn.nRequestAssertionID := 16#6122;
//fbAL1L1.stIn.stBeamParams := PMPS_GVL.cst0RateBeam;
fbAL1L1.stIn.bValid := TRUE;


fbAL1L1(
    stYStage := Main.M1,
    fbArbiter := GVL.fbArbiter1,
    fbFFHWO := GVL.fbFastFaultOutput1);

END_PROGRAM

// ---- POUs/PRG_IM2L1_PPM.TcPOU
PROGRAM PRG_IM2L1_PPM
VAR
        {attribute 'pytmc' := '
        pv: IM2L1:PPM
        io: io
    '}
    {attribute 'TcLinkTo' := '.fbGige.iIlluminatorINT := TIIB[IM2L1-EL4004]^AO Outputs Channel 1^Analog output;
                              .fbGige.bGigePower := TIIB[IM2L1-EL2004]^Channel 3^Output;
                              .fbPowerMeter.iVoltageINT := TIIB[IM2L1-EL3062]^AI Standard Channel 1^Value;
                              .fbPowerMeter.fbThermoCouple.bError := TIIB[IM2L1-EL3314]^TC Inputs Channel 1^Status^Error;
                              .fbPowerMeter.fbThermoCouple.bUnderrange := TIIB[IM2L1-EL3314]^TC Inputs Channel 1^Status^Underrange;
                              .fbPowerMeter.fbThermoCouple.bOverrange := TIIB[IM2L1-EL3314]^TC Inputs Channel 1^Status^Overrange;
                              .fbPowerMeter.fbThermoCouple.iRaw := TIIB[IM2L1-EL3314]^TC Inputs Channel 1^Value;
                              .fbYagThermoCouple.bError := TIIB[IM2L1-EL3314]^TC Inputs Channel 2^Status^Error;
                              .fbYagThermoCouple.bUnderrange := TIIB[IM2L1-EL3314]^TC Inputs Channel 2^Status^Underrange;
                              .fbYagThermoCouple.bOverrange := TIIB[IM2L1-EL3314]^TC Inputs Channel 2^Status^Overrange;
                              .fbYagThermoCouple.iRaw := TIIB[IM2L1-EL3314]^TC Inputs Channel 2^Value'}
    fbIM2L1: FB_PPM;

END_VAR

fbIM2L1.nTransitionAssertionID := 16#2210;
fbIM2L1.nUnknownAssertionID := 16#2219;

fbIM2L1.stOut.fPosition := -8.82;
fbIM2L1.stOut.bUseRawCounts := FALSE;
fbIM2L1.stOut.nRequestAssertionID := 16#2211;
fbIM2L1.stOut.stBeamParams := PMPS_GVL.cstFullBeam;
fbIM2L1.stOut.bValid := TRUE;

fbIM2L1.stPower.fPosition := -47.92;
fbIM2L1.stPower.bUseRawCounts := FALSE;
fbIM2L1.stPower.nRequestAssertionID := 16#2212;
fbIM2L1.stPower.stBeamParams := PMPS_GVL.cstFullBeam;
fbIM2L1.stPower.bValid := TRUE;

fbIM2L1.stYag1.fPosition := -71.92;
fbIM2L1.stYag1.bUseRawCounts := FALSE;
fbIM2L1.stYag1.nRequestAssertionID := 16#2213;
fbIM2L1.stYag1.stBeamParams := PMPS_GVL.cstFullBeam;
fbIM2L1.stYag1.bValid := TRUE;

fbIM2L1.stYag2.fPosition := -94.92;
fbIM2L1.stYag2.bUseRawCounts := FALSE;
fbIM2L1.stYag2.nRequestAssertionID := 16#2214;
fbIM2L1.stYag2.stBeamParams := PMPS_GVL.cstFullBeam;
fbIM2L1.stYag2.bValid := TRUE;

fbIM2L1(
    fbArbiter := GVL.fbArbiter1,
    fbFFHWO := GVL.fbFastFaultOutput1,
    stYStage := Main.M2);

END_PROGRAM

// ---- POUs/PRG_SL3L1_SCATTER.TcPOU
PROGRAM PRG_SL3L1_SCATTER
VAR
    {attribute 'pytmc' := '
        pv: SL3L1:SCATTER
        io: io
    '}
    fbSL3L1: FB_SLITS;
    //GET PMPS Move Ok bit
    // Default True until it is properly linked to PMPS bit
    bMoveOk:BOOL :=TRUE;
    {attribute 'pytmc' := '
    pv: SL3L1:SCATTER:GO;
    io: io;
    field: ZNAM False;
    field: ONAM True;
    '}
    bExecuteMotion :BOOL :=FALSE;
    bTest:BOOL:=FALSE;
    //for testing purposes only. comment-out/delete once done.
    mcPower : ARRAY [1..4] OF MC_POWER;


    (*Offsets*)
    (* Absolute encoder value at the HLS + Absolure eoncoder value at the centered beam *)
    rEncoderOffsetTop: REAL := -15; (* 0+(-15)*)
    rEncoderOffsetBottom: REAL := -15; (* 0+(-15)*)
    rEncoderOffsetNorth: REAL := -15;(* 0+(-15)*)
    rEncoderOffsetSouth: REAL := -15;(* 0+(-15)*)

END_VAR


fbSL3L1.bMoveOk := bMoveOk;

//for testing purposes only. comment-out/delete once done.
If (bTest) THEN
mcPower[1](axis:=Main.M50.Axis, Enable:=bTest, enable_positive:=Main.M50.bLimitForwardEnable, enable_negative:=Main.M50.bLimitBackwardEnable);
mcPower[2](axis:=Main.M51.Axis, Enable:=bTest, enable_positive:=Main.M51.bLimitForwardEnable, enable_negative:=Main.M51.bLimitBackwardEnable);
mcPower[3](axis:=Main.M52.Axis, Enable:=bTest, enable_positive:=Main.M52.bLimitForwardEnable, enable_negative:=Main.M52.bLimitBackwardEnable);
mcPower[4](axis:=Main.M53.Axis, Enable:=bTest, enable_positive:=Main.M53.bLimitForwardEnable, enable_negative:=Main.M53.bLimitBackwardEnable);
ELSE

//Homing routine parameters
Main.M51.fHomePosition:= 0;
Main.M50.fHomePosition:= -30.6;
Main.M52.fHomePosition:= 0;
Main.M53.fHomePosition:= -30.51;

Main.M51.nHomingMode := ENUM_EpicsHomeCmd.HIGH_LIMIT;
Main.M50.nHomingMode := ENUM_EpicsHomeCmd.LOW_LIMIT;
Main.M52.nHomingMode := ENUM_EpicsHomeCmd.HIGH_LIMIT;
Main.M53.nHomingMode := ENUM_EpicsHomeCmd.LOW_LIMIT;


fbSL3L1.rEncoderOffsetTop := rEncoderOffsetTop;
fbSL3L1.rEncoderOffsetBottom := rEncoderOffsetBottom;
fbSL3L1.rEncoderOffsetNorth := rEncoderOffsetNorth;
fbSL3L1.rEncoderOffsetSouth := rEncoderOffsetSouth;

fbSL3L1(stTopBlade:=  Main.M51,
        stBottomBlade:= Main.M50,
        stNorthBlade:=  Main.M52,
        stSouthBlade:=  Main.M53,
        bExecuteMotion:=bExecuteMotion,
        io_fbFFHWO := GVL.fbFastFaultOutput2,
        fbArbiter := GVL.fbArbiter1);

//fbSL3L1.M_CheckPMPS(2);

END_IF

END_PROGRAM

// ---- POUs/PRG_TXI_PM.TcPOU
PROGRAM PRG_TXI_PM
VAR
    {attribute 'pytmc' := '
        pv: TXI:PPM:01
        io: io
    '}
    {attribute 'TcLinkTo' := '.fbPowerMeter.iVoltageINT := TIID^Device 1 (EtherCAT)^TXI Power Meter (EK1100)^PM-EL3064^AI Standard Channel 1^Value'}
    fbTXIPM: FB_PPM;
    dumbymotor : DUT_MotionStage;

END_VAR

fbTXIPM(
    fbArbiter := GVL.fbArbiter1,
    fbFFHWO := GVL.fbFastFaultOutput1,
    stYStage := dumbymotor);

END_PROGRAM

// ---- POUs/PRG_PMPS.TcPOU
PROGRAM PRG_PMPS
VAR
    fbArbiterIO: FB_SubSysToArbiter_IO;
END_VAR

GVL.fbFastFaultOutput1.Execute(i_xVeto := PMPS_GVL.stCurrentBeamParameters.aVetoDevices[PMPS.L_Stopper.ST1L1]);
fbArbiterIO(
    i_bVeto := PMPS_GVL.stCurrentBeamParameters.aVetoDevices[PMPS.L_Stopper.ST1L1],
    Arbiter:=GVL.fbArbiter1,
    fbFFHWO:=GVL.fbFastFaultOutput1);

END_PROGRAM
